// TIA Portal V19 export
TYPE "typePressureGuageRs485ControlNodeCommands"
TITLE = LBC_typeAnalogOutputControlNodeCommands
// Control Node Wapper commands
// stored: Access Published
   STRUCT
      simulation { ExternalAccessible := 'False'; ExternalVisible := 'False'; ExternalWritable := 'False'} : Bool;   // Enable simulation input (process value)
      simulatedAnalogValue { ExternalAccessible := 'False'; ExternalVisible := 'False'; ExternalWritable := 'False'} : Int;   // Input process value for scaling from simulated process
      reset { ExternalAccessible := 'False'; ExternalVisible := 'False'; ExternalWritable := 'False'} : Bool;   // Initialiazing the block TRUE: FB in reset state FALSE: FB in operation
      quality { ExternalAccessible := 'False'; ExternalVisible := 'False'; ExternalWritable := 'False'} : Bool := true;   // Quality bit from sensor FALSE = error, TRUE = healthy [default]
   END_STRUCT;
END_TYPE
